// FB diagnostic and reset 
IF fbJogAcc.Execute AND (NOT fbJogAcc.Busy OR fbJogAcc.InVelocity) THEN
	IF fbJogAcc.Error THEN
		nErrorId := fbJogAcc.ErrorID;
		sLastError := 'Antrieb Tippen Beschleunigung.';
		eState := E_ComponentState.eComponentState_error;
	END_IF
	fbJogAcc.Velocity := 0;
	fbJogAcc.Execute := FALSE;
END_IF

// measure jog time to capture speed at the according ramp positon
tonJogAcc.IN := stJogAccPrm.bJogForward OR stJogAccPrm.bJogBackwards;
tonJogAcc.PT := stJogAccPrm.tAccTime;
tonJogAcc();

// reset jog F/B each cycle (stop's axis if Jog/JogEx method isn't called anymore)
stJogAccPrm.bJogBackwards := FALSE;
stJogAccPrm.bJogForward := FALSE;

IF eCommandExecute <> E_MotionCommand.eMotionCommand_jogAcc THEN
	RETURN;
END_IF

// halt axis if jogAcc timer is disabled
IF NOT tonJogAcc.IN THEN
	fbJogAcc.Velocity := 0;
	eCommandExecute := E_MotionCommand.eMotionCommand_none;
	stHaltPrm.eBufferMode := MC_Aborting;
	stHaltPrm.fDeceleration := stJogAccPrm.fDeceleration;
	stHaltPrm.fJerk := stJogAccPrm.fJerk;
	stHaltPrm.stOptions := stJogAccPrm.stOptions;
	THIS^.HaltEx(stHaltPrm);	
END_IF

sClearText := Concat('Antrieb Tippen Beschleunigung, Geschwindigkeit: ', LREAL_TO_STRING(fbJogAcc.Velocity));
IF fbJogAcc.Velocity < stJogAccPrm.fFastSpeed AND NOT fbJogAcc.Busy THEN
	// ramp = Kx + d
	fbJogAcc.Velocity := (TIME_TO_LREAL(tonJogAcc.ET) * ((stJogAccPrm.fFastSpeed - stJogAccPrm.fSlowSpeed)/TIME_TO_LREAL(tonJogAcc.PT))) + stJogAccPrm.fSlowSpeed;
	// limit speed	
	fbJogAcc.Velocity := LIMIT(stJogAccPrm.fSlowSpeed, fbJogAcc.Velocity, stJogAccPrm.fFastSpeed);
	fbJogAcc(Axis := fbAxisRef, Execute := TRUE);	
END_IF
END_ACTION

ACTION WfMovAbs:

/// Workflow move axis abs

// call fb's cyclic
fbMovAbs1.Position := stMovAbsPrm.fPosition;
fbMovAbs1.Velocity := stMovAbsPrm.fVelocity;
fbMovAbs1.Acceleration := stMovAbsPrm.fAcceleration;
fbMovAbs1.Deceleration := stMovAbsPrm.fDeceleration;
fbMovAbs1.Jerk := stMovAbsPrm.fJerk;
fbMovAbs1.BufferMode := stMovAbsPrm.eBufferMode;
fbMovAbs1.Options := stMovAbsPrm.stOptions;
fbMovAbs1(Axis := fbAxisRef);

fbMovAbs2.Position := stMovAbsPrm.fPosition;
fbMovAbs2.Velocity := stMovAbsPrm.fVelocity;
fbMovAbs2.Acceleration := stMovAbsPrm.fAcceleration;
fbMovAbs2.Deceleration := stMovAbsPrm.fDeceleration;
fbMovAbs2.Jerk := stMovAbsPrm.fJerk;
fbMovAbs2.BufferMode := stMovAbsPrm.eBufferMode;
fbMovAbs2.Options := stMovAbsPrm.stOptions;
fbMovAbs2(Axis := fbAxisRef);

// FB diagnostic and reset 
IF fbMovAbs1.Execute AND NOT fbMovAbs1.Busy THEN
	IF fbMovAbs1.Error THEN
		nErrorId := fbMovAbs1.ErrorID;
		sLastError := 'Antrieb Positionierung Absolut (FB1)';
		eState := E_ComponentState.eComponentState_error;
	END_IF
	fbMovAbs1.Execute := FALSE;
END_IF
IF fbMovAbs2.Execute AND NOT fbMovAbs2.Busy THEN
	IF fbMovAbs2.Error THEN
		nErrorId := fbMovAbs2.ErrorID;
		sLastError := 'Antrieb Positionierung Absolut (FB2)';
		eState := E_ComponentState.eComponentState_error;
	END_IF
	fbMovAbs2.Execute := FALSE;
END_IF

// return if not in move abs
IF eCommandExecute <> E_MotionCommand.eMotionCommand_moveAbs THEN
	RETURN;
END_IF

sClearText := 'Antrieb Positionierung Absolut';		
IF NOT fbMovAbs1.Busy THEN
	fbMovAbs1(Axis := fbAxisRef, Execute := TRUE);
	eCommandExecute := E_MotionCommand.eMotionCommand_none;
ELSIF NOT fbMovAbs2.Busy THEN
	fbMovAbs2(Axis := fbAxisRef, Execute := TRUE);
	eCommandExecute := E_MotionCommand.eMotionCommand_none;
ELSE
	nErrorId := 0;
	sLastError := 'Fehler Antrieb Positionierung Absolut. Kein Baustein bereit';
	eState := E_ComponentState.eComponentState_error;
END_IF
END_ACTION

ACTION WfMovAdd:

/// Workflow move axis add

// call fb's cyclic
fbMovAdd1.Distance := stMovAddPrm.fDistance;
fbMovAdd1.Velocity := stMovAddPrm.fVelocity;
fbMovAdd1.Acceleration := stMovAddPrm.fAcceleration;
fbMovAdd1.Deceleration := stMovAddPrm.fDeceleration;
fbMovAdd1.Jerk := stMovAddPrm.fJerk;
fbMovAdd1.BufferMode := stMovAddPrm.eBufferMode;
fbMovAdd1.Options := stMovAddPrm.stOptions;
fbMovAdd1(Axis := fbAxisRef);

fbMovAdd2.Distance := stMovAddPrm.fDistance;
fbMovAdd2.Velocity := stMovAddPrm.fVelocity;
fbMovAdd2.Acceleration := stMovAddPrm.fAcceleration;
fbMovAdd2.Deceleration := stMovAddPrm.fDeceleration;
fbMovAdd2.Jerk := stMovAddPrm.fJerk;
fbMovAdd2.BufferMode := stMovAddPrm.eBufferMode;
fbMovAdd2.Options := stMovAddPrm.stOptions;
fbMovAdd2(Axis := fbAxisRef);

// FB diagnostic and reset 
IF fbMovAdd1.Execute AND NOT fbMovAdd1.Busy THEN
	IF fbMovAdd1.Error THEN
		nErrorId := fbMovAdd1.ErrorID;
		sLastError := 'Antrieb Positionierung Additiv (FB1)';
		eState := E_ComponentState.eComponentState_error;
	END_IF
	fbMovAdd1.Execute := FALSE;
END_IF
IF fbMovAdd2.Execute AND NOT fbMovAdd2.Busy THEN
	IF fbMovAdd2.Error THEN
		nErrorId := fbMovAdd2.ErrorID;
		sLastError := 'Antrieb Positionierung Additiv (FB2)';
		eState := E_ComponentState.eComponentState_error;
	END_IF
	fbMovAdd2.Execute := FALSE;
END_IF

// return if not in move add
IF eCommandExecute <> E_MotionCommand.eMotionCommand_moveAdd THEN
	RETURN;
END_IF

sClearText := 'Antrieb Positionierung Additiv';
IF NOT fbMovAdd1.Busy THEN
	fbMovAdd1(Axis := fbAxisRef, Execute := TRUE);
	eCommandExecute := E_MotionCommand.eMotionCommand_none;	
ELSIF NOT fbMovAdd2.Busy THEN
	fbMovAdd2(Axis := fbAxisRef, Execute := TRUE);
	eCommandExecute := E_MotionCommand.eMotionCommand_none;	
ELSE
	nErrorId := 0;
	sLastError := 'Fehler Antrieb Positionierung Additiv. Kein Baustein bereit.';
	eState := E_ComponentState.eComponentState_error;
END_IF
END_ACTION

ACTION WfMovMod:

/// Workflow move axis mod

// call fb's cyclic
fbMovMod1.Position := stMovModPrm.fPosition;
fbMovMod1.Direction := stMovModPrm.eDirection;
fbMovMod1.Velocity := stMovModPrm.fVelocity;
fbMovMod1.Acceleration := stMovModPrm.fAcceleration;
fbMovMod1.Deceleration := stMovModPrm.fDeceleration;
fbMovMod1.Jerk := stMovModPrm.fJerk;
fbMovMod1.BufferMode := stMovModPrm.eBufferMode;
fbMovMod1.Options := stMovModPrm.stOptions;
fbMovMod1(Axis := fbAxisRef);

fbMovMod2.Position := stMovModPrm.fPosition;
fbMovMod2.Direction := stMovModPrm.eDirection;
fbMovMod2.Velocity := stMovModPrm.fVelocity;
fbMovMod2.Acceleration := stMovModPrm.fAcceleration;
fbMovMod2.Deceleration := stMovModPrm.fDeceleration;
fbMovMod2.Jerk := stMovModPrm.fJerk;
fbMovMod2.BufferMode := stMovModPrm.eBufferMode;
fbMovMod2.Options := stMovModPrm.stOptions;
fbMovMod2(Axis := fbAxisRef);

// FB diagnostic and reset 
IF fbMovMod1.Execute AND NOT fbMovMod1.Busy THEN
	IF fbMovMod1.Error THEN
		nErrorId := fbMovMod1.ErrorID;
		sLastError := 'Antrieb Positionierung Modulo (FB1)';
		eState := E_ComponentState.eComponentState_error;
	END_IF
	fbMovMod1.Execute := FALSE;
END_IF
IF fbMovMod2.Execute AND NOT fbMovMod2.Busy THEN
	IF fbMovMod2.Error THEN
		nErrorId := fbMovMod2.ErrorID;
		sLastError := 'Antrieb Positionierung Modulo (FB2)';
		eState := E_ComponentState.eComponentState_error;
	END_IF
	fbMovMod2.Execute := FALSE;
END_IF

// return if not in move rel
IF eCommandExecute <> E_MotionCommand.eMotionCommand_moveMod THEN
	RETURN;
END_IF

sClearText := 'Antrieb Positionierung Modulo';		
IF NOT fbMovMod1.Busy THEN
	fbMovMod1(Axis := fbAxisRef, Execute := TRUE);
	eCommandExecute := E_MotionCommand.eMotionCommand_none;
ELSIF NOT fbMovMod2.Busy THEN
	fbMovMod2(Axis := fbAxisRef, Execute := TRUE);
	eCommandExecute := E_MotionCommand.eMotionCommand_none;
ELSE
	nErrorId := 0;
	sLastError := 'Fehler Antrieb Positionierung Modulo. Kein Baustein bereit.';
	eState := E_ComponentState.eComponentState_error;
END_IF
END_ACTION

ACTION WfMovRel:

/// Workflow move axis rel

// call fb's cyclic
fbMovRel1.Distance := stMovRelPrm.fDistance;
fbMovRel1.Velocity := stMovRelPrm.fVelocity;
fbMovRel1.Acceleration := stMovRelPrm.fAcceleration;
fbMovRel1.Deceleration := stMovRelPrm.fDeceleration;
fbMovRel1.Jerk := stMovRelPrm.fJerk;
fbMovRel1.BufferMode := stMovRelPrm.eBufferMode;
fbMovRel1.Options := stMovRelPrm.stOptions;
fbMovRel1(Axis := fbAxisRef);

fbMovRel2.Distance := stMovRelPrm.fDistance;
fbMovRel2.Velocity := stMovRelPrm.fVelocity;
fbMovRel2.Acceleration := stMovRelPrm.fAcceleration;
fbMovRel2.Deceleration := stMovRelPrm.fDeceleration;
fbMovRel2.Jerk := stMovRelPrm.fJerk;
fbMovRel2.BufferMode := stMovRelPrm.eBufferMode;
fbMovRel2.Options := stMovRelPrm.stOptions;
fbMovRel2(Axis := fbAxisRef);

// FB diagnostic and reset 
IF fbMovRel1.Execute AND NOT fbMovRel1.Busy THEN
	IF fbMovRel1.Error THEN
		nErrorId := fbMovRel1.ErrorID;
		sLastError := 'Antrieb Positionierung Relativ (FB1)';
		eState := E_ComponentState.eComponentState_error;
	END_IF
	fbMovRel1.Execute := FALSE;
END_IF
IF fbMovRel2.Execute AND NOT fbMovRel2.Busy THEN
	IF fbMovRel2.Error THEN
		nErrorId := fbMovRel2.ErrorID;
		sLastError := 'Antrieb Positionierung Relativ (FB2)';
		eState := E_ComponentState.eComponentState_error;
	END_IF
	fbMovRel2.Execute := FALSE;
END_IF

// return if not in move rel
IF eCommandExecute <> E_MotionCommand.eMotionCommand_moveRel THEN
	RETURN;
END_IF

sClearText := 'Antrieb Positionierung Relativ';
IF NOT fbMovRel1.Busy THEN
	fbMovRel1(Axis := fbAxisRef, Execute := TRUE);
	eCommandExecute := E_MotionCommand.eMotionCommand_none;	
ELSIF NOT fbMovRel2.Busy THEN
	fbMovRel2(Axis := fbAxisRef, Execute := TRUE);
	eCommandExecute := E_MotionCommand.eMotionCommand_none;	
ELSE
	nErrorId := 0;
	sLastError := 'Fehler Antrieb Positionierung Relativ. Kein Baustein bereit.';
	eState := E_ComponentState.eComponentState_error;
END_IF
END_ACTION

ACTION WfMovVel:

/// Workflow move axis vel

// call fb's cyclic
fbMovVel1.Velocity := stMovVelPrm.fVelocity;
fbMovVel1.Direction := stMovVelPrm.eDirection;
fbMovVel1.Acceleration := stMovVelPrm.fAcceleration;
fbMovVel1.Deceleration := stMovVelPrm.fDeceleration;
fbMovVel1.Jerk := stMovVelPrm.fJerk;
fbMovVel1.BufferMode := stMovVelPrm.eBufferMode;
fbMovVel1.Options := stMovVelPrm.stOptions;
fbMovVel1(Axis := fbAxisRef);

fbMovVel2.Velocity := stMovVelPrm.fVelocity;
fbMovVel2.Direction := stMovVelPrm.eDirection;
fbMovVel2.Acceleration := stMovVelPrm.fAcceleration;
fbMovVel2.Deceleration := stMovVelPrm.fDeceleration;
fbMovVel2.Jerk := stMovVelPrm.fJerk;
fbMovVel2.BufferMode := stMovVelPrm.eBufferMode;
fbMovVel2.Options := stMovVelPrm.stOptions;
fbMovVel2(Axis := fbAxisRef);

// FB diagnostic and reset 
IF fbMovVel1.Execute AND NOT fbMovVel1.Busy THEN
	IF fbMovVel1.Error THEN
		nErrorId := fbMovVel1.ErrorID;
		sLastError := 'Antrieb Konstante Geschwindigkeit (FB1)';
		eState := E_ComponentState.eComponentState_error;
	END_IF
	fbMovVel1.Execute := FALSE;
END_IF
IF fbMovVel2.Execute AND NOT fbMovVel2.Busy THEN
	IF fbMovVel2.Error THEN
		nErrorId := fbMovVel2.ErrorID;
		sLastError := 'Antrieb Konstante Geschwindigkeit (FB2)';
		eState := E_ComponentState.eComponentState_error;
	END_IF
	fbMovVel2.Execute := FALSE;
END_IF

// return if other command active
IF eCommandExecute <> E_MotionCommand.eMotionCommand_moveVel THEN
	RETURN;
END_IF

sClearText := 'Antrieb Konstante Geschwindigkeit';		
IF NOT fbMovVel1.Busy THEN
	fbMovVel1(Axis := fbAxisRef, Execute := TRUE);
	eCommandExecute := E_MotionCommand.eMotionCommand_none;
ELSIF NOT fbMovVel2.Busy THEN
	fbMovVel2(Axis := fbAxisRef, Execute := TRUE);
	eCommandExecute := E_MotionCommand.eMotionCommand_none;
ELSE
	nErrorId := 0;
	sLastError := 'Fehler Antrieb Konstante Geschwindigkeit. Kein Baustein bereit.';
	eState := E_ComponentState.eComponentState_error;
END_IF
END_ACTION

ACTION WfPower:

/// Workflow power axis

tonAutoPowerOff(IN := bEnable AND stDefaultPrm.stGeneralPrm.bEnableAutoPowerOff AND fbAxisRef.Status.NotMoving AND NOT fbAxisRef.Status.Error AND 
					  (eCommandRequest = eMotionCommand_none OR eCommandRequest = eMotionCommand_reset OR eCommandRequest = eMotionCommand_setPos) AND
					  (eCommandExecute = eMotionCommand_none OR eCommandExecute = eMotionCommand_reset OR eCommandExecute = eMotionCommand_setPos),
				PT := stDefaultPrm.stGeneralPrm.tAutoPowerOffDelay);

fbPower.Enable := bEnable AND NOT tonAutoPowerOff.Q;
fbPower(BufferMode := MC_Aborting, Axis := fbAxisRef);

fbPower.Enable_Negative := bEnableNeg AND (NOT bEnableLimit OR stin.bLimitNeg);
fbPower.Enable_Positive := bEnablePos AND (NOT bEnableLimit OR stin.bLimitPos);


// ext. fan control
IF stIn.iMotorTemperature >= stDefaultPrm.stGeneralPrm.iExtFanThreshold THEN
	stOut.bExternalFan := TRUE;
ELSIF stIn.iMotorTemperature < (stDefaultPrm.stGeneralPrm.iExtFanThreshold - 50) THEN // hysteresis 5°C
	stOut.bExternalFan := FALSE;
END_IF
END_ACTION

ACTION WfReset:

/// Workflow resetting

// call FB cyclic
fbReset(Axis:= fbAxisRef);

// FB diagnostic and reset 
IF fbReset.Execute AND NOT fbReset.Busy THEN
	IF fbReset.Error THEN			
		nErrorId := fbReset.ErrorID;
		sLastError := 'Fehler bei Antrieb Reset.';
		eState := E_ComponentState.eComponentState_error;			
	END_IF
	fbReset.Execute := FALSE;
END_IF

// return if other command active
IF eCommandExecute <> E_MotionCommand.eMotionCommand_reset THEN
	RETURN;
END_IF

IF eAxisType = E_AxisType.AX5xxx THEN
	// reset ax5000
	sClearText := 'Start Antrieb Reset';
	IF NOT fbAX5xxxDiag.Busy THEN
		fbAX5xxxDiag.Reset := fbAxisRef.Status.Error OR fbAxisRef.Status.DriveDeviceError;
		eCommandExecute := E_MotionCommand.eMotionCommand_none;
		eState := E_ComponentState.eComponentState_ready;
	END_IF	
ELSE
	// reset sequence of default axis types
	sClearText := 'Start Antrieb Reset';
	IF NOT fbReset.Busy THEN
		fbReset(Axis := fbAxisRef, Execute := fbAxisRef.Status.Error);
		eCommandExecute := E_MotionCommand.eMotionCommand_none;
		eState := E_ComponentState.eComponentState_ready;
	END_IF
END_IF
END_ACTION

ACTION WfSetPos:

/// Workflow set position

// call fb cyclic
fbSetPos.Position := stSetPosPrm.fPosition;
fbSetPos.Mode := stSetPosPrm.bMode;
fbSetPos.Options := stSetPosPrm.stOptions;
fbSetPos(Axis := fbAxisRef);

// FB diagnostic and reset 
IF fbSetPos.Execute AND NOT fbSetPos.Busy THEN
	IF fbSetPos.Error THEN			
		nErrorId := fbSetPos.ErrorID;
		sLastError := 'Fehler Antrieb Position setzen.';
		eState := E_ComponentState.eComponentState_error;			
	END_IF
	fbSetPos.Execute := FALSE;
END_IF

// return if other command active	
IF eCommandExecute <> E_MotionCommand.eMotionCommand_setPos THEN
	RETURN;
END_IF

sClearText := 'ntrieb Position setzen';		
IF NOT fbSetPos.Busy THEN
	fbSetPos(Axis := fbAxisRef, Execute := TRUE);
	eCommandExecute := E_MotionCommand.eMotionCommand_none;
END_IF
END_ACTION

ACTION WfStop:

/// Workflow stopping

// call fb cyclic
fbStop.Deceleration := stStopPrm.fDeceleration;
fbStop.Jerk := stStopPrm.fJerk;
fbStop.Options := stStopPrm.stOptions;
fbStop(Axis := fbAxisRef);

// FB diagnostic and reset
IF fbStop.Execute THEN
	IF fbStop.Error THEN			
		nErrorId := fbStop.ErrorID;
		sLastError := 'Fehler Antrieb Stoppen.';
		eState := E_ComponentState.eComponentState_error;			
	END_IF
	fbStop.Execute := FALSE;
END_IF

// return if other command active
IF eCommandExecute <> E_MotionCommand.eMotionCommand_stop THEN
	RETURN;
END_IF

sClearText := 'Antrieb Stoppen';
fbStop(Axis := fbAxisRef, Execute := TRUE);

// stop command is not auto reset -> ext. reset needed!
(*
IF fbAxisRef.Status.StandStill THEN
	eCommandExecute := E_MotionCommand.eMotionCommand_none;
END_IF
*)
END_ACTION

END_FUNCTION_BLOCK

// ---- BaseComponents/DigitalOutput/FB_DigitalOutput.TcPOU
FUNCTION_BLOCK FB_DigitalOutput EXTENDS FB_ComponentBase
VAR
	/// IO reference
	stOut 					: REFERENCE TO ST_DigitalOutputOut;
	
	fbButton				: FB_sensor;
	
	fbSignal				: FB_TON_RMTH;
	
	tDelay					: TIME;
	
END_VAR

METHOD AutoOff
VAR_INPUT
	Delay					: TIME;
END_VAR
tDelay:= Delay;
END_METHOD

METHOD FB_init : BOOL
VAR_INPUT
	bInitRetains : BOOL; // if TRUE, the retain variables are initialized (warm start / cold start)
	bInCopyCode : BOOL;  // if TRUE, the instance afterwards gets moved into the copy code (online change)
END_VAR
eTyp := E_ComponentType.eComponentType_DigitalOutput;
END_METHOD

PROPERTY OutputState : BOOL
GET
OutputState := stOut.bOutput;
END_GET
END_PROPERTY

METHOD Reset
VAR_INPUT
END_VAR
// base logic run
SUPER^.Reset();

IF NOT __ISVALIDREF(stOut) THEN
	RETURN;
END_IF

stOut.bOutput := FALSE;
END_METHOD

/// Run component logic
{attribute 'object_name' := 'Run'}
METHOD Run : E_ComponentState
VAR_INPUT
END_VAR
// base logic run
Run := SUPER^.Run();

IF NOT __ISVALIDREF(stOut) THEN
	RETURN;
END_IF

fbSignal(in:= stOut.bOutput, pt:=tDelay);

// auto switch off
IF tDelay <> T#0S AND fbSignal.Q THEN
	stOut.bOutput := FALSE;
END_IF
END_METHOD

METHOD SetReferences : E_OperationResult
VAR_IN_OUT
	/// IO structure
	DigitalOutput 		: ST_DigitalOutputIO;
END_VAR
stOut REF= DigitalOutput.stOut;
END_METHOD

METHOD SwitchState
VAR_INPUT
	bEnable				: BOOL;
END_VAR
stout.bOutput := bEnable;
END_METHOD

END_FUNCTION_BLOCK

// ---- Components/MatAndToolHandling/FB_MatAndToolHandling.TcPOU
FUNCTION_BLOCK FB_MatAndToolHandling EXTENDS FB_CompositionBase
VAR
	
	// Sequencer
	fbSeq						: FB_Sequence;
	
	stPosition					: ST_Coordinate;
	nToolDockingNr				: INT;
	
	fVelocityX					: LREAL;	
	fVelocityY					: LREAL;
	fAccelerationX				: LREAL;	
	fAccelerationY				: LREAL;
	
	bJogReverseDirectionX		: BOOL;
	bJogReverseDirectionY		: BOOL;
	bJogX						: BOOL;
	bJogY						: BOOL;
		
	bMoveX						: BOOL;
	bMoveY						: BOOL;
	
	// Watch Variables	
	refObstacle					: REFERENCE TO BOOL;
	bInPosition					: BOOL;
	
	// Tool/Mat Data
	nCurTooldockingNr			: INT;
	afDistanceTooldocking		: ARRAY[1..2] OF REAL;	
	astOffsetDie				: ARRAY[1..2] OF ST_Coordinate;
	

	nVelocityMultiplier			: INT;
	nAccelerationMultiplier		: INT;	
	stOffsetMat					: ST_Coordinate;
	
	
	// Settings
	
	fMaxVelocityX				: LREAL;
	fMinVelocityX				: LREAL;
	fMaxAccelerationX			: LREAL;
	fMinAccelerationX			: LREAL;
	
	fMaxVelocityY				: LREAL;
	fMinVelocityY				: LREAL;
	fMaxAccelerationY			: LREAL;
	fMinAccelerationY			: LREAL;
	
	fDefaultVelocity			: LREAL;
	fDefaultAcceleration		: LREAL;	
	
	fToleranceWindow			: LREAL := 0.5;
	stMaintPosition				: ST_Coordinate;
	
	// Axis
	bEnable						: BOOL := TRUE;
	refEnable					: REFERENCE TO BOOL;
	fbAxisX						: FB_AxisDriver;
	fbAxisY						: FB_AxisDriver;
	
	// Cylinder
	fbToolSelector				: FB_CylinderDriver;
	
END_VAR

METHOD _ChangeTool : BOOL
VAR_INPUT
END_VAR
fbSeq.Name := 'ChangeTool';

CASE fbSeq.Step OF
	

0	 :	fbSeq.StepDefinition('switch Valves for selected Tooldocking', T#0S);
		
		CASE nToolDockingNr OF
			1: fbToolSelector.ToWP();		
			2: fbToolSelector.ToHP();
		END_CASE

		fbSeq.NextStep(10);
	
	
10	 :	fbSeq.StepDefinition('Tooldock changing', T#0S);

		IF fbToolSelector.ActualPosition = fbToolSelector.RequestPosition THEN
			nCurTooldockingNr := nToolDockingNr;
			fbSeq.Finish();
		END_IF
	

END_CASE
END_METHOD

METHOD _Halt : BOOL
VAR_INPUT
END_VAR
fbSeq.Name := 'Halt';

CASE fbSeq.Step OF
	

0	 :	fbSeq.StepDefinition('Punchaxis Halt', T#0S);
		fbAxisX.Halt();
		fbAxisY.Halt();				
		fbSeq.NextStep(10);
	
	
10	 :	fbSeq.StepDefinition('', T#0S);
		IF fbAxisX.NotMoving AND fbAxisY.NotMoving THEN
			fbSeq.Finish();
		END_IF
	
END_CASE
END_METHOD

METHOD _Homeing : BOOL
VAR_INPUT
END_VAR
fbSeq.Name := 'Homeing';

CASE fbSeq.Step OF
	

0	 :	fbSeq.StepDefinition('', T#0S);

		fbSeq.NextStep(10);
	
	
10	 :	fbSeq.StepDefinition('', T#0S);

		fbSeq.NextStep(20);	

		
20	 :	fbSeq.StepDefinition('', T#0S);

		fbSeq.NextStep(30);	

		
30	 :	fbSeq.StepDefinition('', T#0S);

		fbSeq.NextStep(40);

		
40	 :	fbSeq.StepDefinition('', T#0S);

		fbSeq.NextStep(50);

		
50	 :	fbSeq.StepDefinition('', T#0S);

		fbSeq.Finish();

END_CASE
END_METHOD

METHOD _Jog : BOOL
VAR
	
END_VAR
fbSeq.Name := 'Jog';

CASE fbSeq.Step OF
	

0	 :	fbSeq.StepDefinition('Halt Axis', T#0S);
		fbAxisX.Halt();
		fbAxisY.Halt();	
		fbSeq.NextStep(10);
	
10	 :	fbSeq.StepDefinition('Jog Axis', T#0S);
	
		IF bJogX OR bJogY THEN
			fbAxisX.JogAcc(bJogX AND NOT bJogReverseDirectionX , bJogX AND bJogReverseDirectionX);
			fbAxisY.JogAcc(bJogY AND NOT bJogReverseDirectionY , bJogY AND bJogReverseDirectionY);
		ELSE
			fbSeq.NextStep(20);
		END_IF		
		
20	 :	fbSeq.StepDefinition('Jog Finish', T#0S);
		fbAxisX.Halt();
		fbAxisY.Halt();	
		fbSeq.Finish();

END_CASE
END_METHOD

METHOD _MoveAbs : BOOL
VAR
	stMovAbsParameter			: ST_AxisMoveAbsParameter;
END_VAR
fbSeq.Name := 'MoveAbs';

CASE fbSeq.Step OF
	

0	 :	fbSeq.StepDefinition('Move Axis to Position', T#0S);
		
		IF bMoveX THEN
			stMovAbsParameter.fAcceleration := fAccelerationX;
			stMovAbsParameter.fDeceleration := fAccelerationX;
			stMovAbsParameter.fVelocity := fVelocityX;
			stMovAbsParameter.fPosition := stPosition.fX;
			fbAxisX.MoveAbsEx(stMovAbsParameter);
		END_IF
			
		IF bMoveY THEN
			stMovAbsParameter.fAcceleration := fAccelerationY;
			stMovAbsParameter.fDeceleration := fAccelerationY;
			stMovAbsParameter.fVelocity := fVelocityY;
			stMovAbsParameter.fPosition := stPosition.fY;
			fbAxisY.MoveAbsEx(stMovAbsParameter);
		END_IF
		
		fbSeq.NextStep(20);	
		
20	 :	fbSeq.StepDefinition('Axis moving', T#0S);
		IF (fbAxisX.TargetReached(fToleranceWindow) OR NOT bMoveX) AND (fbAxisY.TargetReached(fToleranceWindow) OR NOT bMoveY) THEN
			fbSeq.Finish();
		END_IF

END_CASE
END_METHOD

/// Actual amplifier temp. [°C]
PROPERTY AmplifierTemp : LREAL
GET
/// Actual amplifier temp. [°C]
AmplifierTemp := MAX(fbAxisX.AmplifierTemp, fbAxisY.AmplifierTemp);
END_GET
END_PROPERTY

METHOD ChangeTool : E_OperationResult
VAR_INPUT
	ToolDockingNr				: INT;
END_VAR
// init result pessimistic
ChangeTool := E_OperationResult.eOperationResult_NOk;

bInPosition := FALSE;


stPosition := stMaintPosition;
fVelocityX := fVelocityY := fDefaultVelocity;	
fAccelerationX := fAccelerationY := fDefaultAcceleration;
nToolDockingNr := ToolDockingNr;
bMoveX := TRUE;
bMoveY := TRUE;

fbSeq.Start(E_MatAndToolHandlingCmd.cmdChangeTool);

ChangeTool := E_OperationResult.eOperationResult_Ok;
END_METHOD

PROPERTY CurTool : INT
GET
CurTool := nCurTooldockingNr;
END_GET
END_PROPERTY

METHOD FB_init : BOOL
VAR_INPUT
	bInitRetains : BOOL; // if TRUE, the retain variables are initialized (warm start / cold start)
	bInCopyCode : BOOL;  // if TRUE, the instance afterwards gets moved into the copy code (online change)
END_VAR
eTyp := E_ComponentType.eComponentType_MatAndToolHandling;
END_METHOD

METHOD GetMovementTime : LREAL
VAR_INPUT
	DistanceX		: LREAL;
	DistanceY		: LREAL;
	VelocityX		: LREAL;
	AccelerationX	: LREAL;
	VelocityY		: LREAL;
	AccelerationY	: LREAL;
END_VAR
VAR
	tmpTimeX		: LREAL;
	tmpTimeY		: LREAL;
	
	tmpTimeB		: LREAL;
	tmpTimeBB		: LREAL;
END_VAR
// X
tmpTimeB  := VelocityX/AccelerationX;
tmpTimeBB := 2*SQRT(DistanceX/AccelerationX);

IF tmpTimeBB/2 > tmpTimeB THEN
	tmpTimeX := DistanceX/VelocityX + VelocityX/AccelerationX;
ELSE
	tmpTimeX := tmpTimeBB;
END_IF


// Y
tmpTimeB  := VelocityY/AccelerationY;
tmpTimeBB := 2*SQRT(DistanceY/AccelerationY);

IF tmpTimeBB/2 > tmpTimeB THEN
	tmpTimeY := DistanceY/fVelocityY + VelocityY/AccelerationY;
ELSE
	tmpTimeY := tmpTimeBB;
END_IF


GetMovementTime := MAX(tmpTimeX, tmpTimeY)*1.2;	// 20% sicherheit
END_METHOD

METHOD Halt : E_OperationResult
VAR_INPUT
END_VAR
// init result pessimistic
Halt := E_OperationResult.eOperationResult_NOk;

bInPosition := FALSE;


fVelocityX := fVelocityY := fDefaultVelocity;	
fAccelerationX := fAccelerationY := fDefaultAcceleration;
bMoveX := FALSE;
bMoveY := FALSE;

fbSeq.Start(E_MatAndToolHandlingCmd.cmdHalt);

Halt := E_OperationResult.eOperationResult_Ok;
END_METHOD

PROPERTY Homed : BOOL
GET
Homed := fbaxisX.Homed AND fbaxisY.Homed;
END_GET
END_PROPERTY

METHOD Homing : E_OperationResult
VAR_INPUT
END_VAR
// init result pessimistic
Homing := E_OperationResult.eOperationResult_NOk;

bInPosition := FALSE;


stPosition := stMaintPosition;
fVelocityX := fVelocityY := fDefaultVelocity;	
fAccelerationX := fAccelerationY := fDefaultAcceleration;
bMoveX := TRUE;
bMoveY := TRUE;

fbSeq.Start(E_MatAndToolHandlingCmd.cmdHomeing);

Homing := E_OperationResult.eOperationResult_Ok;
END_METHOD

METHOD JogX : E_OperationResult
VAR_INPUT
	ReverseDirection					: BOOL;
END_VAR
// init result pessimistic
JogX := E_OperationResult.eOperationResult_NOk;
bInPosition := FALSE;

IF fbSeq.SequenceId <> E_MatAndToolHandlingCmd.cmdJog THEN
	fbSeq.Start(E_MatAndToolHandlingCmd.cmdJog);
//	RETURN;
END_IF


bJogReverseDirectionX := ReverseDirection;
bJogX := TRUE;	

JogX := E_OperationResult.eOperationResult_Ok;
END_METHOD

METHOD JogXStop : E_OperationResult
VAR_INPUT
END_VAR
// init result pessimistic
JogXStop := E_OperationResult.eOperationResult_NOk;

bJogX := FALSE;	

JogXStop := E_OperationResult.eOperationResult_Ok;
END_METHOD

METHOD JogY : E_OperationResult
VAR_INPUT
	ReverseDirection					: BOOL;
END_VAR
// init result pessimistic
JogY := E_OperationResult.eOperationResult_NOk;
bInPosition := FALSE;

IF fbSeq.SequenceId <> E_MatAndToolHandlingCmd.cmdJog THEN
	fbSeq.Start(E_MatAndToolHandlingCmd.cmdJog);
//	RETURN;
END_IF


bJogReverseDirectionY := ReverseDirection;
bJogY := TRUE;	

JogY := E_OperationResult.eOperationResult_Ok;
END_METHOD

METHOD JogYStop : E_OperationResult
VAR_INPUT
END_VAR
// init result pessimistic
JogYStop := E_OperationResult.eOperationResult_NOk;

bJogY := FALSE;	

JogYStop := E_OperationResult.eOperationResult_Ok;
END_METHOD

METHOD MaintPos : E_OperationResult
VAR_INPUT
	bXOnly				: BOOL;
	bYOnly				: BOOL;
END_VAR
IF bXOnly THEN
	MaintPos := MoveAbsX(stMaintPosition.fX,fDefaultVelocity, fDefaultAcceleration);	
ELSIF bYOnly THEN
	MaintPos := MoveAbsY(stMaintPosition.fY,fDefaultVelocity, fDefaultAcceleration);
ELSE
	MaintPos := MoveAbs(stMaintPosition,fDefaultVelocity, fDefaultAcceleration,fDefaultVelocity, fDefaultAcceleration);
END_IF


// override the calculated Position, Maintpos is independent of Tool
stPosition := stMaintPosition;
END_METHOD

/// Actual motor temp. [°C]
PROPERTY MotorTemp : LREAL
GET
/// Actual motor temp. [°C]
MotorTemp := MAX(fbAxisX.MotorTemp,fbAxisY.MotorTemp);
END_GET
END_PROPERTY

METHOD MoveAbs : E_OperationResult
VAR_INPUT
	Positon					: ST_Coordinate;
	VelocityX				: LREAL;
	AccelerationX			: LREAL;
	VelocityY				: LREAL;
	AccelerationY			: LREAL;
END_VAR
// init result pessimistic
MoveAbs := E_OperationResult.eOperationResult_NOk;

bInPosition := FALSE;

stPosition.fX := Positon.fX + stOffsetMat.fX ;//+ astOffsetDie[nCurTooldockingNr].fX
stPosition.fY := Positon.fY - afDistanceTooldocking[nCurTooldockingNr] + stOffsetMat.fY; //+ astOffsetDie[nCurTooldockingNr].fY 

// TODO: Check Coordinates if they are in/outside the traversing range

//IF ABS(fbAxisX.ActPos - stPosition.fX) < fToleranceWindow THEN
//	fVelocityY := MAX(MIN(fMaxVelocityY, VelocityY),fMinVelocityY);	
//	fAccelerationY := MAX(MIN(fMaxAccelerationY, AccelerationY),fMinAccelerationY);
//	bMoveX := FALSE;
//	bMoveY := TRUE;	
//ELSIF ABS(fbAxisY.ActPos - stPosition.fY) < fToleranceWindow THEN
//	fVelocityX := MAX(MIN(fMaxVelocityX, VelocityX),fMinVelocityX);	
//	fAccelerationX := MAX(MIN(fMaxAccelerationX, AccelerationX),fMinAccelerationX);
//	bMoveX := TRUE;
//	bMoveY := FALSE;
//ELSE	
	fVelocityY := MAX(MIN(fMaxVelocityY, VelocityY),fMinVelocityY);	
	fAccelerationY := MAX(MIN(fMaxAccelerationY, AccelerationY),fMinAccelerationY);
	fVelocityX := MAX(MIN(fMaxVelocityX, VelocityX),fMinVelocityX);	
	fAccelerationX := MAX(MIN(fMaxAccelerationX, AccelerationX),fMinAccelerationX);
	bMoveX := TRUE;
	bMoveY := TRUE;
	
//END_IF

fbSeq.Start(E_MatAndToolHandlingCmd.cmdMoveAbs);

MoveAbs := E_OperationResult.eOperationResult_Ok;
END_METHOD

METHOD MoveAbsX : E_OperationResult
VAR_INPUT
	Positon					: REAL;
	Velocity				: LREAL;
	Acceleration			: LREAL;
END_VAR
// init result pessimistic
MoveAbsX := E_OperationResult.eOperationResult_NOk;

bInPosition := FALSE;

stPosition := THIS^.Position;
stPosition.fX := Positon;
fVelocityX := MAX(MIN(fMaxVelocityX, Velocity),fMinVelocityX);	
fAccelerationX := MAX(MIN(fMaxAccelerationX, Acceleration),fMinAccelerationX);
bMoveX := TRUE;
bMoveY := FALSE;

fbSeq.Start(E_MatAndToolHandlingCmd.cmdMoveAbs);

MoveAbsX := E_OperationResult.eOperationResult_Ok;
END_METHOD

METHOD MoveAbsY : E_OperationResult
VAR_INPUT
	Positon					: REAL;
	Velocity				: LREAL;
	Acceleration			: LREAL;
END_VAR
// init result pessimistic
MoveAbsY := E_OperationResult.eOperationResult_NOk;

bInPosition := FALSE;

stPosition := THIS^.Position;
stPosition.fY := Positon;
fVelocityY := MAX(MIN(fMaxVelocityY, Velocity),fMinVelocityY);	
fAccelerationY := MAX(MIN(fMaxAccelerationY, Acceleration),fMinAccelerationY);
bMoveX := FALSE;
bMoveY := TRUE;

fbSeq.Start(E_MatAndToolHandlingCmd.cmdMoveAbs);

MoveAbsY := E_OperationResult.eOperationResult_Ok;
END_METHOD

METHOD MoveRelX : E_OperationResult
VAR_INPUT
	Distance				: LREAL;
	Velocity				: LREAL;
	Acceleration			: LREAL;
END_VAR

VAR
	tmpPos					: ST_Coordinate;
END_VAR
// init result pessimistic
MoveRelX := E_OperationResult.eOperationResult_NOk;

bInPosition := FALSE;

tmpPos := Position;
tmpPos.fX := MAX(fbAxisX.LimitNeg, MIN(fbAxisX.LimitPos, tmpPos.fX + Distance));

stPosition := tmpPos;
fVelocityX := MAX(MIN(fMaxVelocityX, Velocity),fMinVelocityX);	
fAccelerationX := MAX(MIN(fMaxAccelerationX, Acceleration),fMinAccelerationX);
bMoveX := TRUE;
bMoveY := FALSE;

fbSeq.Start(E_MatAndToolHandlingCmd.cmdMoveAbs);

MoveRelX := E_OperationResult.eOperationResult_Ok;
END_METHOD

METHOD MoveRelY : E_OperationResult
VAR_INPUT
	Distance				: LREAL;
	Velocity				: LREAL;
	Acceleration			: LREAL;
END_VAR

VAR
	tmpPos					: ST_Coordinate;
END_VAR
// init result pessimistic
MoveRelY := E_OperationResult.eOperationResult_NOk;

bInPosition := FALSE;

tmpPos := Position;
tmpPos.fY := MAX(fbAxisY.LimitNeg, MIN(fbAxisY.LimitPos, tmpPos.fY + Distance));;

stPosition := tmpPos;
fVelocityY := MAX(MIN(fMaxVelocityY, Velocity),fMinVelocityY);	
fAccelerationY := MAX(MIN(fMaxAccelerationY, Acceleration),fMinAccelerationY);
bMoveX := FALSE;
bMoveY := TRUE;

fbSeq.Start(E_MatAndToolHandlingCmd.cmdMoveAbs);

MoveRelY := E_OperationResult.eOperationResult_Ok;
END_METHOD

PROPERTY Moving : BOOL
GET
Moving := fbAxisX.Moving OR fbAxisY.Moving;
END_GET
END_PROPERTY

PROPERTY NotMoving : BOOL
GET
NotMoving := NOT Moving;
END_GET
END_PROPERTY

PROPERTY Override : LREAL
GET
Override := MAX(fbAxisX.Override, fbAxisY.Override);
END_GET
SET
fbAxisX.Override := Override;
fbAxisY.Override := Override;
END_SET
END_PROPERTY

PROPERTY Position : ST_Coordinate
GET
Position.fX := fbAxisX.Position;
Position.fY := fbAxisY.Position;
END_GET
END_PROPERTY

PROPERTY Ready : BOOL
GET
Ready := fbAxisX.MotionState <> MC_AXISSTATE_DISABLED AND fbAxisY.MotionState <> MC_AXISSTATE_DISABLED;
END_GET
END_PROPERTY

/// Reset component logic
{attribute 'object_name' := 'Reset'}
METHOD Reset
// base logic run
SUPER^.Reset();

fbAxisY.Reset();
fbAxisX.Reset();

fbSeq.Init();
END_METHOD

/// Run component logic
{attribute 'object_name' := 'Run'}
METHOD Run : E_ComponentState
// run Base Logic
Run := SUPER^.Run();

IF __ISVALIDREF(refEnable) THEN
	bEnable := refEnable;
END_IF

// run Axis Driver
fbAxisX.Run();
fbAxisX.Enable := bEnable;
fbAxisX.EnablePos := bEnable;
fbAxisX.EnableNeg := bEnable;

fbAxisY.Run();
fbAxisY.Enable := bEnable;
fbAxisY.EnablePos := bEnable;
fbAxisY.EnableNeg := bEnable;

// run Cylinder Driver
fbToolSelector.Run();
fbToolSelector.SafetyOk := bEnable;
fbToolSelector.bEnableHp := bEnable;
fbToolSelector.bEnableWp := bEnable;


// run Sequences
fbSeq.Enable := TRUE;
fbSeq.Base(FALSE, FALSE);
CASE fbSeq.SequenceId OF	
	E_MatAndToolHandlingCmd.cmdMoveAbs:			_MoveAbs();
	E_MatAndToolHandlingCmd.cmdHalt:			_Halt();	
	E_MatAndToolHandlingCmd.cmdChangeTool:		_ChangeTool();	
	E_MatAndToolHandlingCmd.cmdJog:				_Jog();
	E_MatAndToolHandlingCmd.cmdHomeing:			_Homeing();
END_CASE
END_METHOD

METHOD Setup : BOOL
VAR_INPUT
	eAxis_X					: E_Axis;
	eAxis_Y					: E_Axis;
	eToolSelector		    : E_Cylinder;
END_VAR
fbAxisX.Name := 'X-Axis';
fbAxisX.SetAxisReference(COMP.astAxisRef[eAxis_X], COMP.astAxisIO[eAxis_X].stIn, COMP.astAxisIO[eAxis_X].stOut);
fbAxisX.AxisType := E_AxisType.AX5xxx;
fbAxisX.DefaultParameter.stMovAbsPrm.fVelocity := 30;
fbAxisX.Active := TRUE;
fbAxisX.Override := 100;
fbAxisX.DefaultParameter.stJogAccPrm.fFastSpeed := 240;
fbAxisX.DefaultParameter.stJogAccPrm.fSlowSpeed := 10;
fbAxisX.DefaultParameter.stJogAccPrm.tAccTime := T#5S;
fbAxisX.SetSecondPosFeedback(3640, 3.9630466037326388888888888888889E-5);
fbAxisX.EnableLimitSensor:= FALSE;	
fbAxisX.LimitNeg := 10;
fbAxisX.LimitPos := 4070;

fbAxisY.Name := 'Y-Axis';
fbAxisY.SetAxisReference(COMP.astAxisRef[eAxis_Y], COMP.astAxisIO[eAxis_Y].stIn, COMP.astAxisIO[eAxis_Y].stOut);
fbAxisY.AxisType := E_AxisType.AX5xxx;
fbAxisY.DefaultParameter.stMovAbsPrm.fVelocity := 30;
fbAxisY.Active := TRUE;
fbAxisX.Override := 100;
fbAxisY.DefaultParameter.stJogAccPrm.fFastSpeed := 240;
fbAxisY.DefaultParameter.stJogAccPrm.fSlowSpeed := 10;
fbAxisY.DefaultParameter.stJogAccPrm.tAccTime := T#5S;
fbAxisY.EnableLimitSensor:= FALSE;	
fbAxisY.LimitNeg := 5;
fbAxisY.LimitPos := 790;

fbToolSelector.Name := 'Zylinder';
fbToolSelector.SetIoReference(aStCylinderIO[eToolSelector].stIn, aStCylinderIO[eToolSelector].stOut);
fbToolSelector.EnableHpSensor := TRUE;
fbToolSelector.EnableWpSensor := TRUE;
//fbToolSelector.SetImpulseTime := 
//fbToolSelector.PositionValidationTime :=


fMaxVelocityX			:= 4700;
fMinVelocityX			:= 10;
fMaxAccelerationX		:= 10000;
fMinAccelerationX		:= 0;
fMaxVelocityY			:= 3200;
fMinVelocityY			:= 10;
fMaxAccelerationY		:= 10000;
fMinAccelerationY		:= 0;
fDefaultVelocity		:= 100;
fDefaultAcceleration	:= 0;
fToleranceWindow		:= 0.5;
END_METHOD

METHOD SetupEnable : BOOL

VAR_IN_OUT
	bEnable					: BOOL;
END_VAR
refEnable REF= bEnable;
END_METHOD

METHOD SetupMaintPos : BOOL
VAR_INPUT
	MaintPosition		: ST_Coordinate;
END_VAR
stMaintPosition	:=  MaintPosition;
END_METHOD

METHOD SetupMat : BOOL
VAR_INPUT
	Offset			: ST_Coordinate;
END_VAR
stOffsetMat:= Offset;
END_METHOD

METHOD SetupObstacle : BOOL
VAR_IN_OUT
	Obstacle			: BOOL;
END_VAR
refObstacle REF= Obstacle;
END_METHOD

METHOD SetupToolDistance : BOOL
VAR_INPUT
	fDistanceToolDock1		: REAL;
	fDistanceToolDock2		: REAL;
END_VAR
afDistanceTooldocking[1]	:=  fDistanceToolDock1;
afDistanceTooldocking[2]	:=  fDistanceToolDock2;
END_METHOD

METHOD SetupToolholder : BOOL
VAR_INPUT
	DockingNr		: INT;
	fDieOffsetX		: REAL;
	fDieOffsetY		: REAL;
END_VAR
astOffsetDie[DockingNr].fX := fDieOffsetX;
astOffsetDie[DockingNr].fY := fDieOffsetY;
END_METHOD

{attribute 'monitoring' := 'variable'}
PROPERTY TargetReached : BOOL
GET
TargetReached := fbAxisX.TargetReached(fToleranceWindow) AND fbAxisY.TargetReached(fToleranceWindow);
END_GET
END_PROPERTY

PROPERTY ToolChanged : BOOL
GET
ToolChanged := nCurTooldockingNr = nToolDockingNr;
END_GET
END_PROPERTY

/// The torque limit for both directions. [Nm]
PROPERTY TorqueLimitX : LREAL
GET
/// The torque limit for both directions. [1/10%]
TorqueLimitX := fbAxisX.TorqueLimit;
END_GET
SET
fbAxisX.TorqueLimit := TorqueLimitX;
END_SET
END_PROPERTY

/// The torque limit for both directions. [Nm]
PROPERTY TorqueLimitY : LREAL
GET
/// The torque limit for both directions. [1/10%]
TorqueLimitY := fbAxisY.TorqueLimit;
END_GET
SET
fbAxisY.TorqueLimit := TorqueLimitY;
END_SET
END_PROPERTY

END_FUNCTION_BLOCK

// ---- BaseComponents/CylinderDriver/FB_CylinderDriver.TcPOU
FUNCTION_BLOCK PUBLIC FB_CylinderDriver EXTENDS FB_ComponentBase IMPLEMENTS ITF_Cylinder, ITFComponent
VAR_INPUT
	bSafetyOk				: BOOL; // Freigabe von Sicherheit
	
	bEnableHp				: BOOL;	// Freigabe Grundposition
	bEnableWp				: BOOL;	// Freigabe Arbeitsposition
END_VAR
VAR_OUTPUT
	// Zylinder ist in Grundstellung (verzögert)
	bIsInHp	: BOOL;
	// Zylinder ist in Arbeitsstellung (verzögert)
	bIsInWp	: BOOL;
	// Zylinder Ist-Position
	eActPos	: E_CylinderPosition;
END_VAR
VAR
	/// IO reference
	stIn 	: REFERENCE TO ST_CylinderDriverIn;
	stOut 	: REFERENCE TO ST_CylinderDriverOut;
	
	bWpSensor				: BOOL := TRUE;
	bHpSensor				: BOOL := TRUE;
	
	// private var's
	eReqPos					: E_CylinderPosition;	// Zylinder Soll-Position
	fPositionValidationTime	: TIME := T#300MS; 		// Verweilzeit bis die jeweilige Endlage bestätigt wird.
	tImpulseTime 			: TIME := T#0S; 		// Ansteuerzeit für Impulsventile (0 deaktiviert die Impulssteuerung)
	fSupervisionTime		: TIME := T#5S; 		// Verweilzeit nach Ventilansteuerung, bis die Zylinderendlage geprüft wird (0 deaktiviert die Überwachung)
	tonValveChange			: TON;					// Zeit seit Veränderung der Ventilstellung
	tonIsInHp				: TON;					// Verzögerung in Grundstellung
	tonIsInWp				: TON;					// Verzögerung in Arbeitsstellung
END_VAR

///
/// Cylinder driver FB
/// TP/www.rmth.at/06.2015
///

PROPERTY PUBLIC ActualPosition : E_CylinderPosition
GET
ActualPosition := eActPos;
END_GET
END_PROPERTY

PROPERTY PUBLIC EnableHp : BOOL
GET
EnableHp := bEnableHp;
END_GET
SET
bEnableHp := EnableHp;
END_SET
END_PROPERTY

PROPERTY PUBLIC EnableHpSensor : BOOL
GET
EnableHpSensor := bHpSensor;
END_GET
SET
bHpSensor := EnableHpSensor;
END_SET
END_PROPERTY

PROPERTY PUBLIC EnableWp : BOOL
GET
EnableWp := bEnableWp;
END_GET
SET
bEnableWp := EnableWp;
END_SET
END_PROPERTY

PROPERTY PUBLIC EnableWpSensor : BOOL
GET
EnableWpSensor := bWpSensor;
END_GET
SET
bWpSensor := EnableWpSensor;
END_SET
END_PROPERTY

METHOD FB_init : BOOL
VAR_INPUT
	bInitRetains : BOOL; // if TRUE, the retain variables are initialized (warm start / cold start)
	bInCopyCode : BOOL;  // if TRUE, the instance afterwards gets moved into the copy code (online change)
END_VAR
eTyp := E_ComponentType.eComponentType_Cylinder;
END_METHOD

// Ansteuerzeit für Impulsventile (0 deaktiviert die Impulssteuerung)
PROPERTY PUBLIC ImpulseTime : TIME
GET
// Ansteuerzeit für Impulsventile (0 deaktiviert die Impulssteuerung)
ImpulseTime := tImpulseTime;
END_GET
SET
// Ansteuerzeit für Impulsventile (0 deaktiviert die Impulssteuerung)
tImpulseTime := ImpulseTime;
END_SET
END_PROPERTY

/// Verweilzeit bis die jeweilige Endlage bestätigt wird.
PROPERTY PUBLIC PositionValidationTime : TIME
GET
/// Verweilzeit bis die jeweilige Endlage bestätigt wird.
PositionValidationTime := fPositionValidationTime;
END_GET
SET
/// Verweilzeit bis die jeweilige Endlage bestätigt wird.
fPositionValidationTime := PositionValidationTime;
END_SET
END_PROPERTY

PROPERTY PUBLIC RequestPosition : E_CylinderPosition
GET
RequestPosition := eReqPos;
END_GET
END_PROPERTY

METHOD Reset
VAR_INPUT
END_VAR
// base logic run
SUPER^.Reset();

//ToHP();
tonValveChange(IN := FALSE);
tonIsInHp(IN := FALSE);
tonIsInWp(IN := FALSE);

eState := E_ComponentState.eComponentState_ready;
END_METHOD

METHOD PUBLIC ResetValves
VAR_INPUT
END_VAR
IF NOT __ISVALIDREF(stOut) THEN
	sLastError := 'IO reference not set';
	eState := E_ComponentState.eComponentState_error;
	RETURN;
END_IF

// chk
IF NOT bSafetyOk THEN
	sClearText := 'Warte auf Sicherheit Ok';
	RETURN;
END_IF

eReqPos := eCylinderPosition_unknown;
stOut.bValveCylinderHp := FALSE;
stOut.bValveCylinderWp := FALSE;
tonValveChange(IN := FALSE);
END_METHOD

/// Run component logic
{attribute 'object_name' := 'Run'}
METHOD Run : E_ComponentState
// base logic run
Run := SUPER^.Run();

// chk
IF NOT (__ISVALIDREF(stIn) AND __ISVALIDREF(stOut)) THEN
	sLastError := 'IO reference not set';
	eState := E_ComponentState.eComponentState_error;
	RETURN;
END_IF



// definiere aktuelle Zylinderposition
IF (stIn.bCylinderSensorHp OR (NOT bHpSensor AND stOut.bValveCylinderHp)) AND NOT stIn.bCylinderSensorWp THEN
	eActPos := eCylinderPosition_hp;
ELSIF NOT stIn.bCylinderSensorHp AND (stIn.bCylinderSensorWp OR (NOT bWpSensor AND stOut.bValveCylinderWp)) THEN
	eActPos := eCylinderPosition_wp;
ELSE
	eActPos := eCylinderPosition_unknown;
END_IF

tonIsInHp(IN := (eActPos = eCylinderPosition_hp), PT := fPositionValidationTime);
bIsInHp := tonIsInHp.Q;

tonIsInWp(IN := (eActPos = eCylinderPosition_wp), PT := fPositionValidationTime);
bIsInWp := tonIsInWp.Q;

// Zeitmessung seit Veränderung der Ventilstellung 
tonValveChange(IN := TRUE, PT := tMaxTime);

// für Impulsventile (T#0S od. Wartungsmodus -> Funktion deaktiv)
IF tImpulseTime > T#0S AND tonValveChange.ET > tImpulseTime THEN
	stOut.bValveCylinderHp := FALSE;
	stOut.bValveCylinderWp := FALSE;
END_IF

// Zylinderüberwachung (T#0S -> Funktion deaktiv)
IF fSupervisionTime > T#0S AND tonValveChange.ET > fSupervisionTime AND eActPos <> eReqPos THEN
	IF eReqPos = eCylinderPosition_hp THEN
		sLastError := Concat(sName, ' Grundstellung nicht erreicht.');
		IF stIn.bCylinderSensorWp THEN
			sLastError := Concat(sLastError, ' Signal Arbeitsstellung steht noch an.');
		END_IF
		IF NOT stIn.bCylinderSensorHp THEN
			sLastError := Concat(sLastError, ' Signal Sensor Grundstellung fehlt.');
		END_IF
		IF __ISVALIDREF(fbEventLog) THEN		
			WriteError(E_Event.eEvent_none , sLastError);	
		END_IF
		eState := E_ComponentState.eComponentState_error;
	ELSIF eReqPos = eCylinderPosition_wp THEN
		sLastError := Concat(sName, ' Arbeitsstellung nicht erreicht.');
		IF stIn.bCylinderSensorHp THEN
			sLastError := Concat(sLastError, ' Signal Grundstellung steht noch an.');
		END_IF
		IF NOT stIn.bCylinderSensorWp THEN
			sLastError := Concat(sLastError, ' Signal Arbeitsstellung fehlt.');
		END_IF
		IF __ISVALIDREF(fbEventLog) THEN
			WriteError(E_Event.eEvent_none , sLastError);
		END_IF
		eState := E_ComponentState.eComponentState_error;
	END_IF
END_IF

//
END_METHOD

PROPERTY PUBLIC SafetyOk : BOOL
GET
SafetyOk := bSafetyOk;
END_GET
SET
bSafetyOk := SafetyOk;
END_SET
END_PROPERTY

PROPERTY PUBLIC SensorHp : BOOL
GET
IF __ISVALIDREF(stIn) THEN
	SensorHp := stIn.bCylinderSensorHp;
END_IF
END_GET
END_PROPERTY

PROPERTY PUBLIC SensorWp : BOOL
GET
IF __ISVALIDREF(stIn) THEN
	SensorWp := stIn.bCylinderSensorWp;
END_IF
END_GET
END_PROPERTY

METHOD PUBLIC SetImpulseTime
VAR_INPUT
	/// Ansteuerzeit für Impulsventile (0 deaktiviert die Impulssteuerung)
	tTime : TIME;
END_VAR
END_METHOD

/// Set up reference dependencies.
{attribute 'object_name' := 'SetIoReference'}
METHOD SetIoReference
VAR_IN_OUT
	stRefIn		: ST_CylinderDriverIn;
	stRefOut	: ST_CylinderDriverOut;
END_VAR
stIn 	REF= stRefIn;
stOut 	REF= stRefOut;
END_METHOD

/// Verweilzeit nach Ventilansteuerung, bis die Zylinderendlage geprüft wird (0 deaktiviert die Überwachung)
PROPERTY PUBLIC SupervisionTime : TIME
GET
/// Verweilzeit nach Ventilansteuerung, bis die Zylinderendlage geprüft wird (0 deaktiviert die Überwachung)
SupervisionTime := fSupervisionTime;
END_GET
SET
/// Verweilzeit nach Ventilansteuerung, bis die Zylinderendlage geprüft wird (0 deaktiviert die Überwachung)
fSupervisionTime := SupervisionTime;
END_SET
END_PROPERTY

METHOD PUBLIC ToHP
VAR_INPUT
END_VAR
IF NOT __ISVALIDREF(stOut) THEN
	sLastError := 'IO reference not set';
	eState := E_ComponentState.eComponentState_error;
	RETURN;
END_IF

// chk
IF NOT bSafetyOk THEN
	sClearText := 'Warte auf Sicherheit Ok';
	RETURN;
ELSIF NOT bEnableHp THEN
	sClearText := 'Warte auf Freigabe Hp';
	RETURN;
END_IF

eReqPos := eCylinderPosition_hp;
stOut.bValveCylinderHp := TRUE;
stOut.bValveCylinderWp := FALSE;
tonValveChange(IN := FALSE);
END_METHOD

METHOD PUBLIC ToWP
VAR_INPUT
END_VAR
IF NOT __ISVALIDREF(stOut) THEN
	sLastError := 'IO reference not set';
	eState := E_ComponentState.eComponentState_error;
	RETURN;
END_IF

// chk
IF NOT bSafetyOk THEN
	sClearText := 'Warte auf Sicherheit Ok';
	RETURN;
ELSIF NOT bEnableWp THEN
	sClearText := 'Warte auf Freigabe WP';
	RETURN;
END_IF

eReqPos := eCylinderPosition_wp;
stOut.bValveCylinderHp := FALSE;
stOut.bValveCylinderWp := TRUE;
tonValveChange(IN := FALSE);
END_METHOD

END_FUNCTION_BLOCK

// ---- BaseComponents/AxisDriver/Utilities/FB_AxisDistanceTrigger.TcPOU
FUNCTION_BLOCK FB_AxisDistanceTrigger
VAR_INPUT
	/// reset FB
	bReset: BOOL;
	/// actual position
	fActualPos: LREAL;
	/// trigger distance
	fTriggerDistance: LREAL;
END_VAR
VAR_OUTPUT
	/// trigger output
	Q: BOOL;
END_VAR
VAR
	/// distance
	fDistance: LREAL;
	/// actual ABS position
	fActualAbsPos: LREAL;
	/// mirror ABS position
	fMirrorAbsPos: LREAL;
	bInit: BOOL;
END_VAR
VAR CONSTANT
	fEpsilon: LREAL := 0.01;
END_VAR

fActualAbsPos:=ABS(fActualPos);

IF bReset OR NOT bInit THEN
	bInit:=TRUE;
	Q:=FALSE;
	fMirrorAbsPos:=fActualAbsPos;
	IF bReset THEN	
		fDistance:=0;
	END_IF

END_IF

IF fTriggerDistance <= 0 THEN
	Q:=FALSE;
	RETURN;
END_IF

IF ABS(fActualAbsPos - fMirrorAbsPos) > fEpsilon THEN
	fDistance:=fDistance + ABS(fActualAbsPos - fMirrorAbsPos);
	fMirrorAbsPos:=fActualAbsPos;
END_IF

Q:=fDistance>=fTriggerDistance;

END_FUNCTION_BLOCK

// ---- BaseComponents/AxisDriver/Utilities/FB_LimitSwitchRefSim.TcPOU
/// Axis driver limit switch
FUNCTION_BLOCK FB_LimitSwitchRefSim
VAR_INPUT
	/// Aktiviert die Logik
	bEnable					:BOOL;
	/// Position der Achse
	fPosition				:REAL;
	
	/// Endschalter (Oeffner)
	bLimitSwitch			:BOOL;
	/// Distanz Simuliertem Ref-Schalter zu Endschalter
	fRefLimitDistance		:REAL := 1;
	
	/// Referenzposition
	fRefPosition			:REAL;
	/// Pruefen des Positionsbereichs der Referenzposition
	fRefPosCheckArea		:REAL := 0.2;
END_VAR
VAR_OUTPUT
	/// Endschalter (Verzeogert)
	bLimitSwitchSim			:BOOL;
	/// Simulierter Ref Schalter
	bRefSwitchSim			:BOOL;
	
	/// Pruefung der Refpos OK
	bRefCheckOk				:BOOL;
END_VAR
VAR
	
END_VAR
VAR PERSISTENT
	fPosLatched			:REAL;
	bPosLatched			:BOOL;
END_VAR

(*
	Baustein um einen Ref-Schalter und Limitswitch mit 1 Eingang zu realisieren
	RE / 2015 / www.rmth.at
*)

IF NOT bEnable THEN
	bLimitSwitchSim := bLimitSwitch;
	bRefSwitchSim := bLimitSwitchSim;
	bRefCheckOk := FALSE;
	RETURN;
END_IF

// logik
IF bLimitSwitch THEN // (Oeffner)
	fPosLatched := 0;
	bPosLatched := FALSE;	
	bLimitSwitchSim := TRUE; // limit ok
	bRefSwitchSim := FALSE; // kein referenz

ELSE
	// Position merken
	IF NOT bPosLatched THEN
		bPosLatched := TRUE;
		fPosLatched := fPosition;
	END_IF

	bRefSwitchSim := TRUE;
	bLimitSwitchSim := (ABS(fPosition - fPosLatched) >= fRefLimitDistance);
END_IF

// Referenzpunkt pruefen
bRefCheckOk := ABS(fRefPosition - fPosLatched) <= fRefPosCheckArea;

METHOD Reset : bool
VAR_INPUT
END_VAR
fPosLatched := 0;
bPosLatched := FALSE;
END_METHOD

END_FUNCTION_BLOCK

// ---- BaseComponents/AxisDriver/Utilities/F_LRealToString.TcPOU
FUNCTION F_LRealToString : STRING(255)
VAR_INPUT
	fValue: LREAL;
END_VAR

F_LRealToString := F_LRealToStringEx(fValue, 3);

END_FUNCTION

// ---- BaseComponents/AxisDriver/Utilities/F_LRealToStringEx.TcPOU
FUNCTION F_LRealToStringEx : STRING(255)
VAR_INPUT
	fValue: LREAL;
	iPrecision: INT := 3;
END_VAR
VAR
	fbFormat: FB_FormatString;
END_VAR

fbFormat( sFormat := Concat3('%.', INT_TO_STRING(iPrecision), 'f'), arg1 := F_LREAL( fValue ), sOut => F_LRealToStringEx);

END_FUNCTION

// ---- BaseComponents/AxisDriver/Utilities/F_SpeedReached.TcPOU
/// determines whether the actual speed (ABS value) is within the target-speed window
FUNCTION F_SpeedReached : BOOL
VAR_INPUT
	/// actual speed
	fActualSpeed: LREAL;
	/// target speed
	fTargetSpeed: LREAL;
	/// Override for axis and spindle
	fOverride: LREAL;
END_VAR

F_SpeedReached := F_SpeedWindowReached(fToleranceFactor:=0, fActualSpeed:=fActualSpeed, fTargetSpeed:=fTargetSpeed, fOverride:=fOverride);

END_FUNCTION

// ---- BaseComponents/AxisDriver/Utilities/F_SpeedWindowReached.TcPOU
/// determines whether the actual speed (ABS value) is within the target-speed window
FUNCTION F_SpeedWindowReached : BOOL
VAR_INPUT
	/// factor for tolerance (default: 0.1)
	fToleranceFactor: REAL;
	/// actual speed
	fActualSpeed: LREAL;
	/// target speed
	fTargetSpeed: LREAL;
	/// Override for axis and spindle
	fOverride: LREAL;
END_VAR
VAR CONSTANT
	fDefaultfToleranceFactor: REAL := 0.1;
END_VAR
VAR
	fTol: LREAL;
	fMin: LREAL;
	fMax: LREAL;
	fAct: LREAL;
	fTar: LREAL;
END_VAR

// validate tolerance factor
IF fToleranceFactor <= 0 THEN
	fToleranceFactor:=fDefaultfToleranceFactor;
END_IF

// calc tolerance window and ABS values
fTar:=fTargetSpeed*(fOverride/100);
fTol:=ABS(fTar) * fToleranceFactor;
fMin:=ABS(fTar) - fTol;
fMax:=ABS(fTar) + fTol;
fAct:=ABS(fActualSpeed);

F_SpeedWindowReached := fAct >= fMin AND fAct <= fMax;

END_FUNCTION

// ---- BaseComponents/AxisDriver/Utilities/F_TargetReached.TcPOU
FUNCTION F_TargetReached : BOOL
VAR_INPUT
	fCurrentPos: LREAL;
	fTargetPos: LREAL;
END_VAR


F_TargetReached := F_TargetWindowReached(fCurrentPos, fTargetPos, fEpsilon);

END_FUNCTION

// ---- BaseComponents/AxisDriver/Utilities/F_TargetWindowReached.TcPOU
FUNCTION F_TargetWindowReached : BOOL
VAR_INPUT
	fCurrentPos: LREAL;
	fTargetPos: LREAL;
	fWindow: LREAL;
END_VAR


F_TargetWindowReached := fCurrentPos >= (fTargetPos - fWindow) AND fCurrentPos <= (fTargetPos + fWindow);

END_FUNCTION

// ---- BaseComponents/AxisDriver/Utilities/F_TargetReachedOrHigher.TcPOU
FUNCTION F_TargetReachedOrHigher : BOOL
VAR_INPUT
	fCurrentPos: LREAL;
	fTargetPos: LREAL;
END_VAR


F_TargetReachedOrHigher := fCurrentPos >= (fTargetPos - fEpsilon);

END_FUNCTION

// ---- BaseComponents/AxisDriver/Utilities/F_TargetReachedOrLower.TcPOU
FUNCTION F_TargetReachedOrLower : BOOL
VAR_INPUT
	fCurrentPos: LREAL;
	fTargetPos: LREAL;
END_VAR


F_TargetReachedOrLower := fCurrentPos <= (fTargetPos + fEpsilon);

END_FUNCTION

// ---- BaseComponents/AxisDriver/Utilities/F_TargetWindowReachedAxisRef.TcPOU
FUNCTION F_TargetWindowReachedAxisRef : BOOL
VAR_IN_OUT
	/// Achse als Referenz
	fbAxis		:FB_AxisDriver;
END_VAR
VAR_INPUT
	fTargetPos: LREAL;
	fWindow: LREAL;
END_VAR


F_TargetWindowReachedAxisRef := fbAxis.Position >= (fTargetPos - fWindow) AND fbAxis.Position <= (fTargetPos + fWindow);

END_FUNCTION

// ---- BaseComponents/DigitalInput/FB_DigitalInput.TcPOU
FUNCTION_BLOCK FB_DigitalInput EXTENDS FB_ComponentBase
VAR
	/// IO reference
	stIn 					: REFERENCE TO ST_DigitalInputIn;
	tOnTime					: DT;
	tOffTime				: DT;
	
	fbSensor				: FB_sensor;
END_VAR

PROPERTY Delayed : BOOL
GET
Delayed := fbSensor.Q;
END_GET
END_PROPERTY

PROPERTY ElapsedTime : TIME
GET
ElapsedTime := DT_TO_TIME(tOffTime) - DT_TO_TIME(tOntime);
END_GET
END_PROPERTY

PROPERTY Falling : BOOL
GET
Falling := fbSensor.Qf;
END_GET
END_PROPERTY

METHOD FB_init : BOOL
VAR_INPUT
	bInitRetains : BOOL; // if TRUE, the retain variables are initialized (warm start / cold start)
	bInCopyCode : BOOL;  // if TRUE, the instance afterwards gets moved into the copy code (online change)
END_VAR
eTyp := E_ComponentType.eComponentType_DigitalSensor;
END_METHOD

PROPERTY Raising : BOOL
GET
Raising := fbSensor.Qr;
END_GET
END_PROPERTY

METHOD Reset
VAR_INPUT
END_VAR
// base logic run
SUPER^.Reset();
END_METHOD

/// Run component logic
{attribute 'object_name' := 'Run'}
METHOD Run : E_ComponentState
VAR_INPUT
END_VAR
// base logic run
Run := SUPER^.Run();

fbSensor(b_Signal := stIn.bSensor);

IF fbSensor.Qr THEN
	tOnTime := statics.dtNow;	
	tOffTime := statics.dtNow;
END_IF

IF fbSensor.Qf THEN
	tOffTime := statics.dtNow;
END_IF
END_METHOD

METHOD SetReferences : E_OperationResult
VAR_IN_OUT
	/// IO structure
	DigitalInput 		: ST_DigitalInputIn;
END_VAR
stIn REF= DigitalInput;
END_METHOD

PROPERTY Signal : BOOL
GET
Signal := fbSensor.b_Signal;
END_GET
END_PROPERTY

END_FUNCTION_BLOCK

// ---- BaseComponents/EtherCAT/FB_EtherCatBox.TcPOU
FUNCTION_BLOCK FB_EtherCatBox EXTENDS FB_ComponentBase
VAR
	/// IO structure
	stIO 				: REFERENCE TO ST_EtherCatBoxIO;
	oldEtherCatBoxState : INT;
END_VAR

///
/// EtherCATBox driver.
/// Hannes Fuger / asma.at / 12.2015
///

METHOD FB_init : BOOL
VAR_INPUT
	bInitRetains : BOOL; // if TRUE, the retain variables are initialized (warm start / cold start)
	bInCopyCode : BOOL;  // if TRUE, the instance afterwards gets moved into the copy code (online change)
END_VAR
eTyp := E_ComponentType.eComponentType_EtherCATBox;
END_METHOD

METHOD Run : E_ComponentState
VAR_INPUT
END_VAR
// base logic run
Run := SUPER^.Run();

// chk reference
IF NOT __ISVALIDREF(fbEventLog) THEN
	RETURN;
END_IF

// chk Box name
IF sName = sEmpty THEN
	RETURN;
END_IF

IF oldEtherCatBoxState = stIo.aeEtherCatBoxState THEN
	RETURN;
ELSE
	oldEtherCatBoxState := stIo.aeEtherCatBoxState;
END_IF

// switch state 
CASE stIo.aeEtherCatBoxState OF
	// 0x___1 = Slave in 'INIT' state
	eEtherCatSlaveState_INIT:
		WriteError(eEvent_EcSlaveError , Concat3(sName, ' EcState: ', '0x___1 = Slave in "INIT" state'));
		
	// 0x___2 = Slave in 'PREOP' state
	eEtherCatSlaveState_PREOP:
		WriteError(eEvent_EcSlaveError , Concat3(sName, ' EcState: ', '0x___2 = Slave in "PREOP" state'));
		
	// 0x___3 = Slave in 'BOOT' state
	eEtherCatSlaveState_BOOT:
		WriteError(eEvent_EcSlaveError , Concat3(sName, ' EcState: ', '0x___3 = Slave in "BOOT" state'));
		
	// 0x___4 = Slave in 'SAFEOP' state
	eEtherCatSlaveState_SAFEOP:
		WriteError(eEvent_EcSlaveError , Concat3(sName, ' EcState: ', '0x___4 = Slave in "SAFEOP" state'));
		
	// 0x___8 = Slave in 'OP' state
	eEtherCatSlaveState_OP:
		//fbHMI.SetNotificationPrio(eNotification_EcSlaveInfo, Concat3(sBoxName, ' EcState: ', '0x___8 = Slave in "OP" state'), E_Priority.ePriority_info);
		
	// 0x001_ = Slave signals error
	eEtherCatSlaveState_SignalsError:
		WriteError(eEvent_EcSlaveError , Concat3(sName, ' EcState: ', '0x001_ = Slave signals error'));
		
	// 0x002_ = Invalid vendorId, productCode... read
	eEtherCatSlaveState_Invalid:
		WriteError(eEvent_EcSlaveError , Concat3(sName, ' EcState: ', '0x002_ = Invalid vendorId, productCode... read'));
		
	// 0x004_ = Initialization error occurred
	eEtherCatSlaveState_InitErr:
		WriteError(eEvent_EcSlaveError , Concat3(sName, ' EcState: ', '0x004_ = Initialization error occurred'));
		
	// 0x008_ = Slave disabled
	eEtherCatSlaveState_Disabled:
		WriteError(eEvent_EcSlaveError , Concat3(sName, ' EcState: ', '0x008_ = Slave disabled'));
		
	// 0x010_ = Slave not present
	eEtherCatSlaveState_NotPresent:
		WriteError(eEvent_EcSlaveError , Concat3(sName, ' EcState: ', '0x010_ = Slave not present'));
		
	// 0x020_ = Slave signals link error
	eEtherCatSlaveState_LinkErr:
		WriteError(eEvent_EcSlaveError , Concat3(sName, ' EcState: ', '0x020_ = Slave signals link error'));
		
	// 0x040_ = Slave signals missing link
	eEtherCatSlaveState_MissingLink:
		WriteError(eEvent_EcSlaveError , Concat3(sName, ' EcState: ', '0x040_ = Slave signals missing link'));
		
	// 0x080_ = Slave signals unexpected link
	eEtherCatSlaveState_UnexpectedLink:
		WriteError(eEvent_EcSlaveError , Concat3(sName, ' EcState: ', '0x080_ = Slave signals unexpected link'));
		
	// 0x100_ = Communication port A
	eEtherCatSlaveState_ComPortA:
		WriteError(eEvent_EcSlaveError , Concat3(sName, ' EcState: ', '0x100_ = Communication port A'));
		                                                                                              
	// 0x200_ = Communication port B                                                                  
	eEtherCatSlaveState_ComPortB:                                                                     
		WriteError(eEvent_EcSlaveError , Concat3(sName, ' EcState: ', '0x200_ = Communication port B'));
		                                                                                              
	// 0x400_ = Communication port C                                                                  
	eEtherCatSlaveState_ComPortC:                                                                     
		WriteError(eEvent_EcSlaveError , Concat3(sName, ' EcState: ', '0x400_ = Communication port C'));
		                                                                                              
	// 0x800_ = Communication port D                                                                  
	eEtherCatSlaveState_ComPortD:                                                                     
		WriteError(eEvent_EcSlaveError , Concat3(sName, ' EcState: ', '0x800_ = Communication port D'));
		
ELSE
	IF stIo.aeEtherCatBoxState <> eEtherCatSlaveState_OP THEN
		WriteError(eEvent_EcSlaveError , Concat3(sName, ': EcState ', INT_TO_STRING(stIo.aeEtherCatBoxState)));
	END_IF
END_CASE
END_METHOD

/// Dependency injection method.
{attribute 'object_name' := 'SetReferences'}
METHOD SetReferences
VAR_IN_OUT
	/// IO structure
	stRefIO		: ST_EtherCatBoxIO;
END_VAR
/// set up references
stIO REF= stRefIO;
END_METHOD

END_FUNCTION_BLOCK

// ---- BaseComponents/Supervision/CheckFunctions/CheckBounds.TcPOU
/// Implicitly generated code : DO NOT EDIT!!!
/// CheckBounds is used to check for range overflows
{attribute 'check_bounds' := ''}
{attribute 'no_check' := ''}
FUNCTION CheckBounds : DINT
VAR_INPUT
	index: DINT;
	lower: DINT;
	upper: DINT;
END_VAR

// align bounds 
CheckBounds := MIN(upper, MAX(lower, index));

// if index changed, report error
IF CheckBounds <> index THEN
	GVL_Supervision.aCodeErr[eCodeError_bounds] := TRUE;
END_IF

END_FUNCTION

// ---- BaseComponents/Supervision/CheckFunctions/CheckDivDInt.TcPOU
/// Implicitly generated code : DO NOT EDIT!!!
/// Checks for division by 0, if divisor is 0, replace it with 1 and report error
{attribute 'check_div_int32' := ''}
{attribute 'no_check' := ''}
FUNCTION CheckDivDInt : DINT
VAR_INPUT
	divisor: DINT;
END_VAR

IF divisor = 0 THEN
	// replace divisor and report error if necessary
	CheckDivDInt := 1;
	GVL_Supervision.aCodeErr[eCodeError_divDInt] := TRUE;
ELSE
	CheckDivDInt := divisor;
END_IF;

END_FUNCTION

// ---- BaseComponents/Supervision/CheckFunctions/CheckDivLInt.TcPOU
/// Implicitly generated code : DO NOT EDIT!!!
/// Checks for division by 0, if divisor is 0, replace it with 1 and report error
{attribute 'no_check' := ''}
{attribute 'check_div_int64' := ''}
FUNCTION CheckDivLInt : LINT
VAR_INPUT
	divisor: LINT;
END_VAR

IF divisor = 0 THEN
	// replace divisor and report error if necessary
	CheckDivLInt := 1;
	GVL_Supervision.aCodeErr[eCodeError_divLInt] := TRUE;
ELSE
	CheckDivLInt := divisor;
END_IF;

END_FUNCTION

// ---- BaseComponents/Supervision/CheckFunctions/CheckDivLReal.TcPOU
/// Implicitly generated code : DO NOT EDIT!!!
/// Checks for division by 0, if divisor is 0, replace it with 1 and report error
{attribute 'no_check' := ''}
{attribute 'check_div_real64' := ''}
FUNCTION CheckDivLReal : LREAL
VAR_INPUT
	divisor: LREAL;
END_VAR

IF divisor = 0 THEN
	// replace divisor and report error if necessary
	CheckDivLReal := 1;
	GVL_Supervision.aCodeErr[eCodeError_divLReal] := TRUE;
ELSE
	CheckDivLReal:=divisor;
END_IF;

END_FUNCTION

// ---- BaseComponents/Supervision/CheckFunctions/CheckDivReal.TcPOU
/// Implicitly generated code : DO NOT EDIT
/// Checks for division by 0, if divisor is 0, replace it with 1 and report error
{attribute 'check_div_real32' := ''}
{attribute 'no_check' := ''}
FUNCTION CheckDivReal : REAL
VAR_INPUT
	divisor: REAL;
END_VAR

IF divisor = 0 THEN
	// replace divisor and report error if necessary
	CheckDivReal := 1;
	GVL_Supervision.aCodeErr[eCodeError_divReal] := TRUE;
ELSE
	CheckDivReal := divisor;
END_IF;

END_FUNCTION

// ---- BaseComponents/Supervision/CheckFunctions/CheckPointer.TcPOU
/// Implicitly generated code : DO NOT EDIT!!!
/// checks for correct pointer use. Currently, this only detects null pointer, which are replaced by 
/// a pointer to a dummy area and reported as error
{attribute 'check_pointer' := ''}
{attribute 'no_check' := ''}
FUNCTION CheckPointer : POINTER TO BYTE
VAR_INPUT
	/// Destination address of the pointer
	ptToTest: POINTER TO BYTE;
	/// Size of the type the pointer points to. (e.g: 20 for POINTER TO ARRAY [0..9] OF INT) 
	iSize: DINT;
	/// Granularity of the pointer access. This is the size of the biggest non-structured data type in the type the pointer points to. (e.g: 2 for POINTER TO ARRAY [0..9] OF INT)
	iGran: DINT;
	/// Indicates read or write Access. TRUE = write access.
	bWrite: BOOL;
END_VAR

VAR_STAT
	aDummyData						: ARRAY[0..1023] OF BYTE;	
END_VAR

// check for outside address range
IF ptToTest = 0 THEN
	// report error 
	GVL_Supervision.aCodeErr[eCodeError_pointer] := TRUE;
	// this is just a desparate way to keep the PLC from crashing, 
	// probably there's a better solution
	CheckPointer := ADR( aDummyData ); 
END_IF

END_FUNCTION

// ---- BaseComponents/Supervision/CheckFunctions/CheckRangeSigned.TcPOU
/// Implicitly generated code : DO NOT EDIT!!!
/// Checks subrange value. If value is outside [lower,upper], it is set to the closer bound and reports the error.
{attribute 'check_range_signed' := ''}
{attribute 'no_check' := ''}
FUNCTION CheckRangeSigned : DINT
VAR_INPUT
	value: DINT;
	lower: DINT;
	upper: DINT;
END_VAR

// align to bounds 
CheckRangeSigned := MIN( upper, MAX( lower, value ));

// if value changed, report error
IF CheckRangeSigned <> value THEN
	GVL_Supervision.aCodeErr[eCodeError_rangeSigned] := TRUE;
END_IF

END_FUNCTION

// ---- BaseComponents/Supervision/CheckFunctions/CheckRangeUnsigned.TcPOU
/// Implicitly generated code : DO NOT EDIT
/// Checks subrange value. If value is outside [lower,upper], it is set to the closer bound and reports the error.
{attribute 'check_range_unsigned' := ''}
{attribute 'no_check' := ''}
FUNCTION CheckRangeUnsigned : UDINT
VAR_INPUT
	value: UDINT;
	lower: UDINT;
	upper: UDINT;
END_VAR

// align to bounds 
CheckRangeUnsigned := MIN(upper, MAX(lower, value));

// if value changed, report error
IF CheckRangeUnsigned <> value THEN
	GVL_Supervision.aCodeErr[eCodeError_rangeUnsigned] := TRUE;
END_IF

END_FUNCTION

// ---- Utilities/TaskAllocation/P_Fast.TcPOU
/// Fast Task program
PROGRAM P_Fast
VAR CONSTANT
	iMaxTaskAllocation				: INT := 10;
END_VAR

VAR
	ii	: INT;
	aItfTasks						: ARRAY[0..255] OF ITF_TaskAllocation;	  
END_VAR

/// run cyclic fast tasks
FOR ii := 0 TO iMaxTaskAllocation DO
	IF aItfTasks[ii] = 0 THEN
		CONTINUE;
	END_IF
	IF aItfTasks[ii].Task = E_Task.eTask_fast THEN
		aItfTasks[ii].Invoke();
	END_IF
END_FOR

METHOD RegisterTask : E_OperationResult
VAR_INPUT
	/// Task to be registered
	ITask	: ITF_TaskAllocation;
END_VAR
VAR
	ii	: INT;
END_VAR
/// queue task
FOR ii := 0 TO iMaxTaskAllocation DO
	IF aItfTasks[ii] <> 0 THEN
		IF aItfTasks[ii].TaskId <> ITask.TaskId THEN
			CONTINUE;
		END_IF
	END_IF
	ITask.TaskId := ii + 1;
	aItfTasks[ii] := ITask;
	EXIT;
END_FOR
END_METHOD

METHOD UnregisterTask : E_OperationResult
VAR_INPUT
	/// Task to be unregistered
	ITask	: ITF_TaskAllocation;
END_VAR
VAR
	ii	: INT;
END_VAR
/// dequeue task
FOR ii := 0 TO iMaxTaskAllocation DO
	IF aItfTasks[ii] = 0 THEN
		CONTINUE;
	END_IF
	IF aItfTasks[ii].TaskId <> ITask.TaskId THEN
		CONTINUE;
	END_IF
	aItfTasks[ii] := 0;
END_FOR
END_METHOD

END_PROGRAM
